Universal Robots PolyScope program: test_read_xyz.urp

Program test_read_xyz (installation=default directory=/ursim/programs createdIn=3.15.8.106339 lastSavedIn=3.15.8.106339 robotSerialNumber=2018359999)
Calibrated DH parameters: a=[0, -0.425, -0.39225, 0, 0, 0]; d=[0.089159, 0, 0, 0.10915, 0.09465, 0.0823]; alpha=[1.570796, 0, 0, 1.570796, -1.570796, 0]; deltaTheta=[0, 0, 0, 0, 0, 0]
BeforeStart
  time_count := 0
  temp_joint := [0,0,0,0,0,0]
  target_joint := p[0,0,0,0,0,0]
  data_recv_len := 6
  host := "127.0.0.1"
  port_no := 12345
  open := socket_open(host, port_no)
  Loop While (checkContinuously=false) expression=open≟False
    open := socket_open(host, port_no)
  target_pos := p[0,0,0,0,3.14,0]
  counter := 0
Robot Program (runOnlyOnce=false)
  send_to_server := "send_to_server"
  Script: socket_send_string(send_to_server)
  recv_from_serv := socket_read_ascii_float(data_recv_len)
  Loop While (checkContinuously=false) expression=recv_from_serv[0]≠data_recv_len
    recv_from_serv := socket_read_ascii_float(data_recv_len)
  Loop While (checkContinuously=false) expression=counter < data_recv_len
    Script: target_pos[counter]=recv_from_serv[counter+1]
    counter := counter+1
  counter := 0
  Script: movej(get_inverse_kin(target_pos))
  Script: sync()
Thread Thread_1 (runOnlyOnce=false)
  Script: time_count=time_count+1
  time_sec := time_count / 125
  Script: sync()
